TYPE StatsAggregateFIFOBuffer :
STRUCT
	Size: UDINT := 864; (*3 days at 5 min*)
	Buffer: ARRAY [0..863] OF StatsAggregateRecord;
END_STRUCT
END_TYPE

(* stored: Version 1.1.0.1, ProductVersion 3.1.4024.9
   DUT StatsAggregateFIFOBuffer: Id {2210022f-e07a-430f-92be-b0e2ec571d96} *)
